(* CODESYS project MotorSequence.xml

Project tree, tasks and I/O mapping:
  function block MotorSequence [LD]
*)

// MotorSequence
FUNCTION_BLOCK MotorSequence
VAR_INPUT
	CommandForward: BOOL;
	CommandReverse: BOOL;
	Stop: BOOL;
	ForwardTarget: BOOL;
	ReverseTarget: BOOL;
	Reset: BOOL; // To reset after complete.
	BrakeOffDelay: TIME;
	MotorOnDelay: TIME;
	MotorOffDelay: TIME;
	BrakeOnDelay: TIME;
	MinimumDuration: TIME;
	MaximumDuration: TIME;
	
END_VAR
VAR_OUTPUT
	Executing: BOOL;
	AtForward: BOOL;
	AtReverse: BOOL;
	Forward: BOOL;
	Reverse: BOOL;
	Brake: BOOL;
	Fault: BOOL; // Outputs True if any Fault present.
	TimeoutFault: BOOL; // Outputs True if the motor running time exceeds the timeout input setting.
	DirectionFault: BOOL; // Outputs True if the opposite sensor is reached after the minimum time setting.	
END_VAR
VAR
	_ForwardRS: RS;
	_ReverseRS: RS;
	
	_ExecutingForward: BOOL;
	_ExecutingReverse: BOOL;
	
	_AtForwardRS: RS;
	_AtReverseRS: RS;
	
	_TargetReachedRS: RS;
	_TargetReached: BOOL;
	
	_MotorOn: TON;
	_MotorOff: TON;
	_BrakeOn: TON;
	_BrakeOff: TON;
	
	_MinimumDurationTimer: TON;
	_MaximumDurationTimer: TON;	
	_CompleteRS: RS;
	_ExecutingRS: RS;
	_StopExecuting: BOOL;
	_SequenceComplete: BOOL;
	_MaximumDurationRS: RS;
	//_MinimumDurationRS: RS;
	_DirectionFaultRS: RS;
END_VAR
VAR // added by the converter: edge detectors and wires of the graphical bodies
    _rt1, _rt2, _rt3 : R_TRIG;
END_VAR

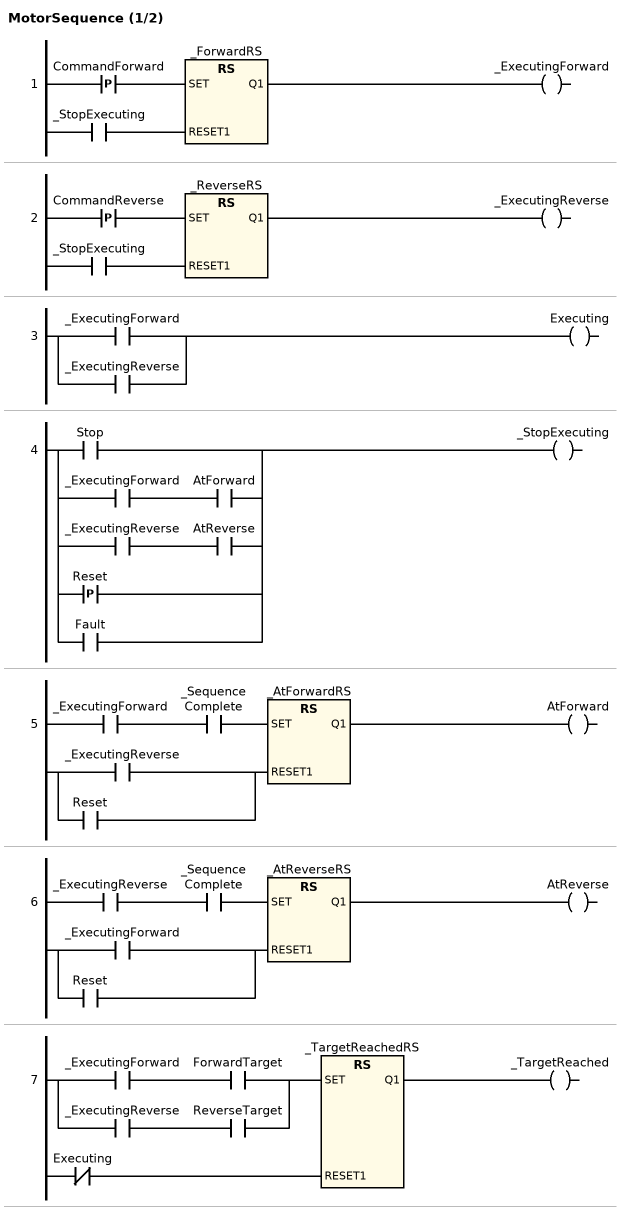
// NETWORK 1
_rt1(CLK := CommandForward);
_ForwardRS(SET := _rt1.Q, RESET1 := _StopExecuting); // RS
_ExecutingForward := _ForwardRS.Q1;

// NETWORK 2
_rt2(CLK := CommandReverse);
_ReverseRS(SET := _rt2.Q, RESET1 := _StopExecuting); // RS
_ExecutingReverse := _ReverseRS.Q1;

// NETWORK 3
Executing := _ExecutingForward OR _ExecutingReverse;

// NETWORK 4
_rt3(CLK := Reset);
_StopExecuting := Stop OR _ExecutingForward AND AtForward OR _ExecutingReverse AND AtReverse OR _rt3.Q OR Fault;

// NETWORK 5
_AtForwardRS(SET := _ExecutingForward AND _SequenceComplete, RESET1 := _ExecutingReverse OR Reset); // RS
AtForward := _AtForwardRS.Q1;

// NETWORK 6
_AtReverseRS(SET := _ExecutingReverse AND _SequenceComplete, RESET1 := _ExecutingForward OR Reset); // RS
AtReverse := _AtReverseRS.Q1;

// NETWORK 7
_TargetReachedRS(SET := _ExecutingForward AND ForwardTarget OR _ExecutingReverse AND ReverseTarget, RESET1 := NOT Executing); // RS
_TargetReached := _TargetReachedRS.Q1;

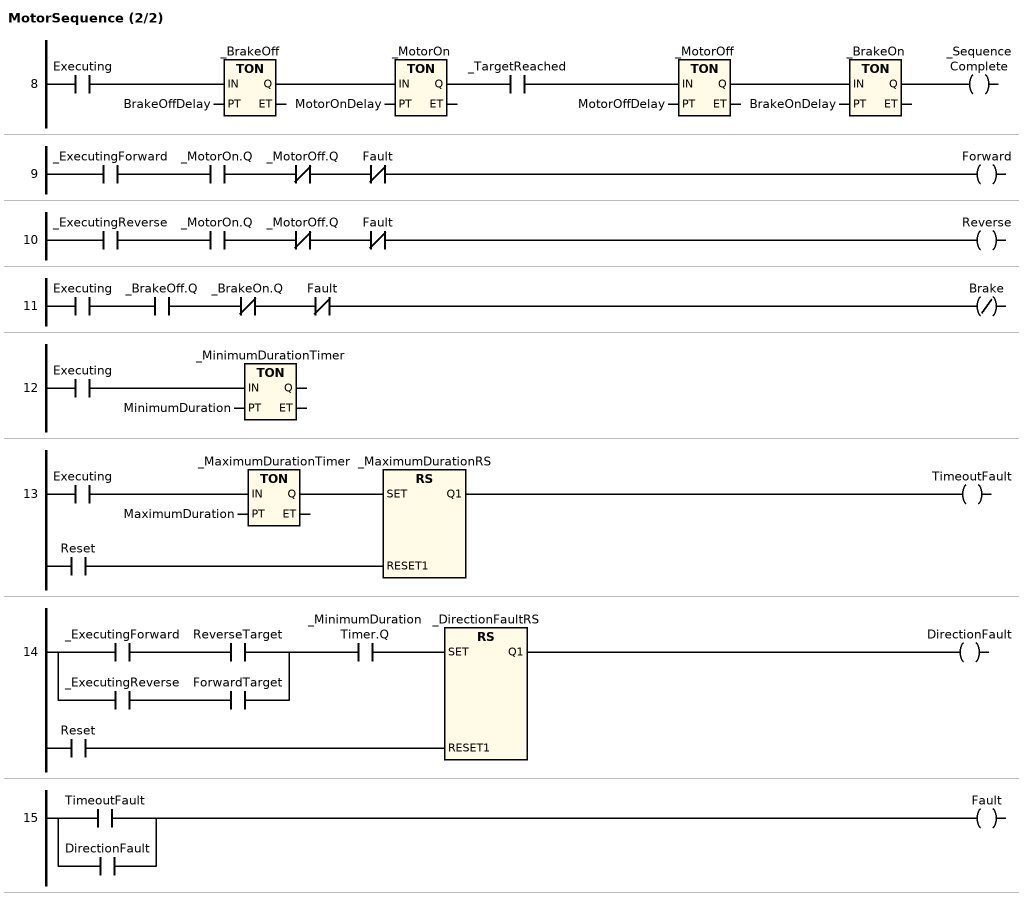
// NETWORK 8
_BrakeOff(IN := Executing, PT := BrakeOffDelay); // TON
_MotorOn(IN := _BrakeOff.Q, PT := MotorOnDelay); // TON
_MotorOff(IN := _MotorOn.Q AND _TargetReached, PT := MotorOffDelay); // TON
_BrakeOn(IN := _MotorOff.Q, PT := BrakeOnDelay); // TON
_SequenceComplete := _BrakeOn.Q;

// NETWORK 9
Forward := _ExecutingForward AND _MotorOn.Q AND NOT _MotorOff.Q AND NOT Fault;

// NETWORK 10
Reverse := _ExecutingReverse AND _MotorOn.Q AND NOT _MotorOff.Q AND NOT Fault;

// NETWORK 11
Brake := NOT (Executing AND _BrakeOff.Q AND NOT _BrakeOn.Q AND NOT Fault);

// NETWORK 12
_MinimumDurationTimer(IN := Executing, PT := MinimumDuration); // TON

// NETWORK 13
_MaximumDurationTimer(IN := Executing, PT := MaximumDuration); // TON
_MaximumDurationRS(SET := _MaximumDurationTimer.Q, RESET1 := Reset); // RS
TimeoutFault := _MaximumDurationRS.Q1;

// NETWORK 14
_DirectionFaultRS(SET := (_ExecutingForward AND ReverseTarget OR _ExecutingReverse AND ForwardTarget) AND _MinimumDurationTimer.Q, RESET1 := Reset); // RS
DirectionFault := _DirectionFaultRS.Q1;

// NETWORK 15
Fault := TimeoutFault OR DirectionFault;

END_FUNCTION_BLOCK
